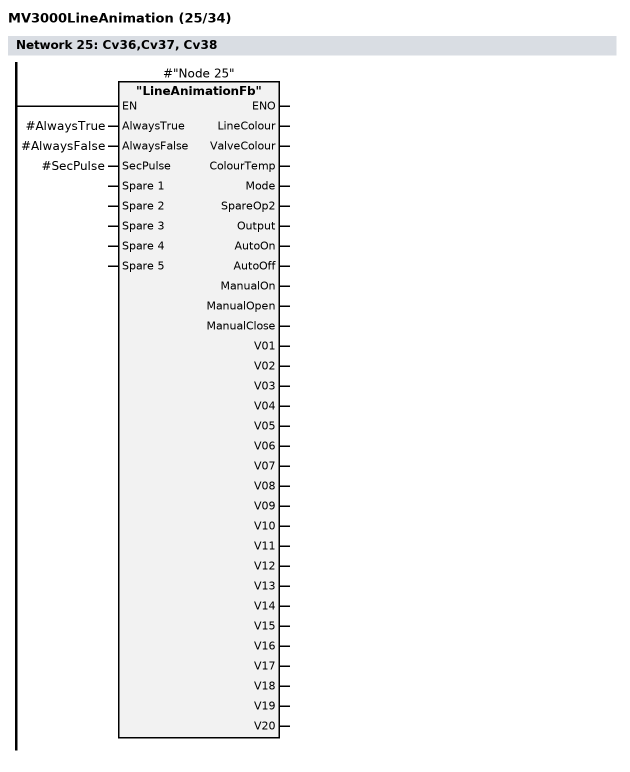
   RUNG wire#powerrail
      #"Node 25"(AlwaysTrue := #AlwaysTrue, AlwaysFalse := #AlwaysFalse, SecPulse := #SecPulse, "Spare 1" :=, "Spare 2" :=, "Spare 3" :=, "Spare 4" :=, "Spare 5" :=, LineColour =>, ValveColour =>, ColourTemp =>, Mode =>, SpareOp2 =>, Output =>, AutoOn =>, AutoOff =>, ManualOn =>, ManualOpen =>, ManualClose =>, V01 =>, V02 =>, V03 =>, V04 =>, V05 =>, V06 =>, V07 =>, V08 =>, V09 =>, V10 =>, V11 =>, V12 =>, V13 =>, V14 =>, V15 =>, V16 =>, V17 =>, V18 =>, V19 =>, V20 =>)
   END_RUNG
   // the same network as SCL:
   #"Node 25"(AlwaysTrue := #AlwaysTrue, AlwaysFalse := #AlwaysFalse, SecPulse := #SecPulse);   // "LineAnimationFb"
END_REGION

REGION Network 26: Cv30,Cv33, Cv34,Cv35
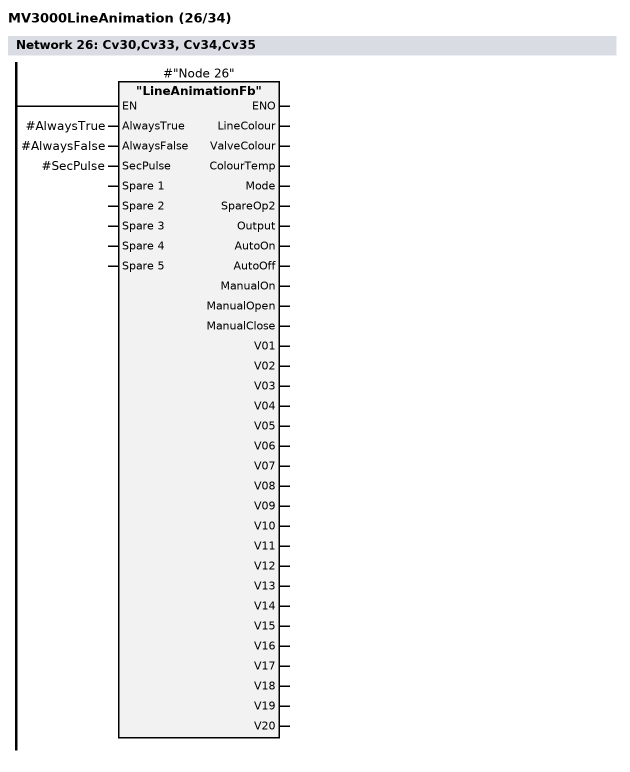
   RUNG wire#powerrail
      #"Node 26"(AlwaysTrue := #AlwaysTrue, AlwaysFalse := #AlwaysFalse, SecPulse := #SecPulse, "Spare 1" :=, "Spare 2" :=, "Spare 3" :=, "Spare 4" :=, "Spare 5" :=, LineColour =>, ValveColour =>, ColourTemp =>, Mode =>, SpareOp2 =>, Output =>, AutoOn =>, AutoOff =>, ManualOn =>, ManualOpen =>, ManualClose =>, V01 =>, V02 =>, V03 =>, V04 =>, V05 =>, V06 =>, V07 =>, V08 =>, V09 =>, V10 =>, V11 =>, V12 =>, V13 =>, V14 =>, V15 =>, V16 =>, V17 =>, V18 =>, V19 =>, V20 =>)
   END_RUNG
   // the same network as SCL:
   #"Node 26"(AlwaysTrue := #AlwaysTrue, AlwaysFalse := #AlwaysFalse, SecPulse := #SecPulse);   // "LineAnimationFb"
END_REGION

REGION Network 27: Cv28, Cv34,Cv37,Cv45,Cv51, Cv57,Cv60
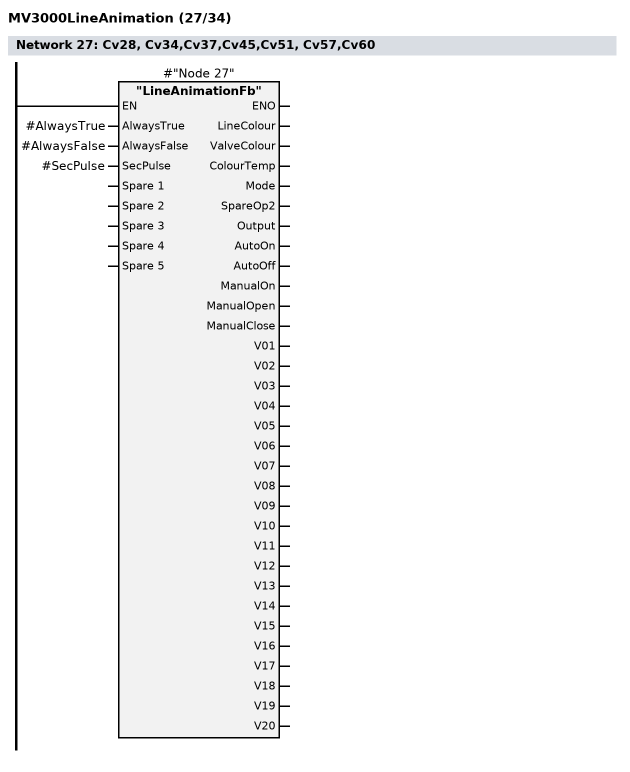
   RUNG wire#powerrail
      #"Node 27"(AlwaysTrue := #AlwaysTrue, AlwaysFalse := #AlwaysFalse, SecPulse := #SecPulse, "Spare 1" :=, "Spare 2" :=, "Spare 3" :=, "Spare 4" :=, "Spare 5" :=, LineColour =>, ValveColour =>, ColourTemp =>, Mode =>, SpareOp2 =>, Output =>, AutoOn =>, AutoOff =>, ManualOn =>, ManualOpen =>, ManualClose =>, V01 =>, V02 =>, V03 =>, V04 =>, V05 =>, V06 =>, V07 =>, V08 =>, V09 =>, V10 =>, V11 =>, V12 =>, V13 =>, V14 =>, V15 =>, V16 =>, V17 =>, V18 =>, V19 =>, V20 =>)
   END_RUNG
   // the same network as SCL:
   #"Node 27"(AlwaysTrue := #AlwaysTrue, AlwaysFalse := #AlwaysFalse, SecPulse := #SecPulse);   // "LineAnimationFb"
END_REGION

REGION Network 28: Cv22, Cv25,Cv19,Cv20,Cv29,Cv35, Cv38,C46 ,Cv52 ,Cv58 ,Cv59
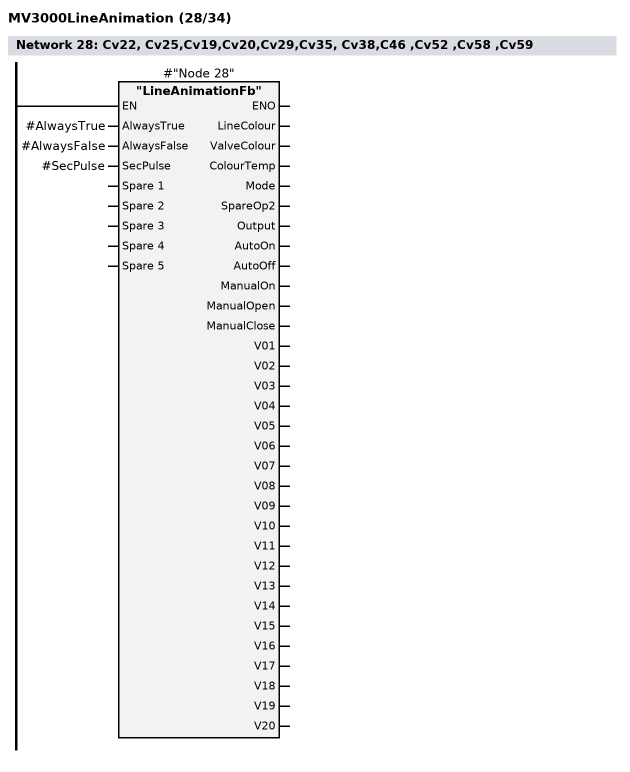
   RUNG wire#powerrail
      #"Node 28"(AlwaysTrue := #AlwaysTrue, AlwaysFalse := #AlwaysFalse, SecPulse := #SecPulse, "Spare 1" :=, "Spare 2" :=, "Spare 3" :=, "Spare 4" :=, "Spare 5" :=, LineColour =>, ValveColour =>, ColourTemp =>, Mode =>, SpareOp2 =>, Output =>, AutoOn =>, AutoOff =>, ManualOn =>, ManualOpen =>, ManualClose =>, V01 =>, V02 =>, V03 =>, V04 =>, V05 =>, V06 =>, V07 =>, V08 =>, V09 =>, V10 =>, V11 =>, V12 =>, V13 =>, V14 =>, V15 =>, V16 =>, V17 =>, V18 =>, V19 =>, V20 =>)
   END_RUNG
   // the same network as SCL:
   #"Node 28"(AlwaysTrue := #AlwaysTrue, AlwaysFalse := #AlwaysFalse, SecPulse := #SecPulse);   // "LineAnimationFb"
END_REGION

REGION Network 29: Cv01,Cv04
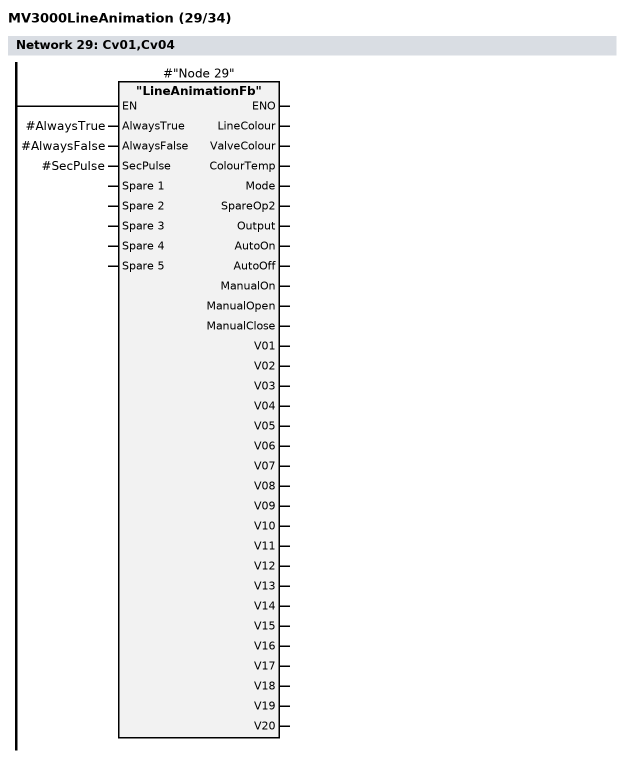
   RUNG wire#powerrail
      #"Node 29"(AlwaysTrue := #AlwaysTrue, AlwaysFalse := #AlwaysFalse, SecPulse := #SecPulse, "Spare 1" :=, "Spare 2" :=, "Spare 3" :=, "Spare 4" :=, "Spare 5" :=, LineColour =>, ValveColour =>, ColourTemp =>, Mode =>, SpareOp2 =>, Output =>, AutoOn =>, AutoOff =>, ManualOn =>, ManualOpen =>, ManualClose =>, V01 =>, V02 =>, V03 =>, V04 =>, V05 =>, V06 =>, V07 =>, V08 =>, V09 =>, V10 =>, V11 =>, V12 =>, V13 =>, V14 =>, V15 =>, V16 =>, V17 =>, V18 =>, V19 =>, V20 =>)
   END_RUNG
   // the same network as SCL:
   #"Node 29"(AlwaysTrue := #AlwaysTrue, AlwaysFalse := #AlwaysFalse, SecPulse := #SecPulse);   // "LineAnimationFb"
END_REGION

REGION Network 30: Cv06,Cv09
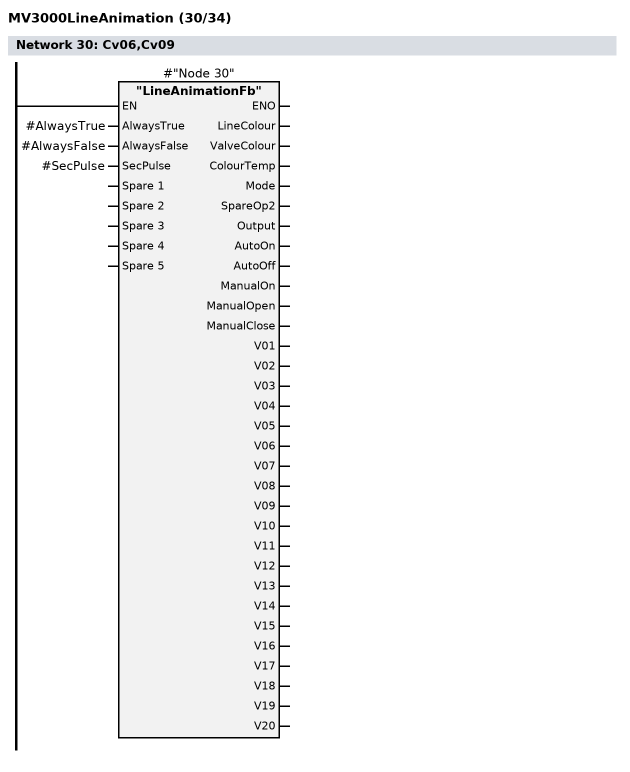
   RUNG wire#powerrail
      #"Node 30"(AlwaysTrue := #AlwaysTrue, AlwaysFalse := #AlwaysFalse, SecPulse := #SecPulse, "Spare 1" :=, "Spare 2" :=, "Spare 3" :=, "Spare 4" :=, "Spare 5" :=, LineColour =>, ValveColour =>, ColourTemp =>, Mode =>, SpareOp2 =>, Output =>, AutoOn =>, AutoOff =>, ManualOn =>, ManualOpen =>, ManualClose =>, V01 =>, V02 =>, V03 =>, V04 =>, V05 =>, V06 =>, V07 =>, V08 =>, V09 =>, V10 =>, V11 =>, V12 =>, V13 =>, V14 =>, V15 =>, V16 =>, V17 =>, V18 =>, V19 =>, V20 =>)
   END_RUNG
   // the same network as SCL:
   #"Node 30"(AlwaysTrue := #AlwaysTrue, AlwaysFalse := #AlwaysFalse, SecPulse := #SecPulse);   // "LineAnimationFb"
END_REGION

REGION Network 31: Cv06,Cv09 ,Cv08
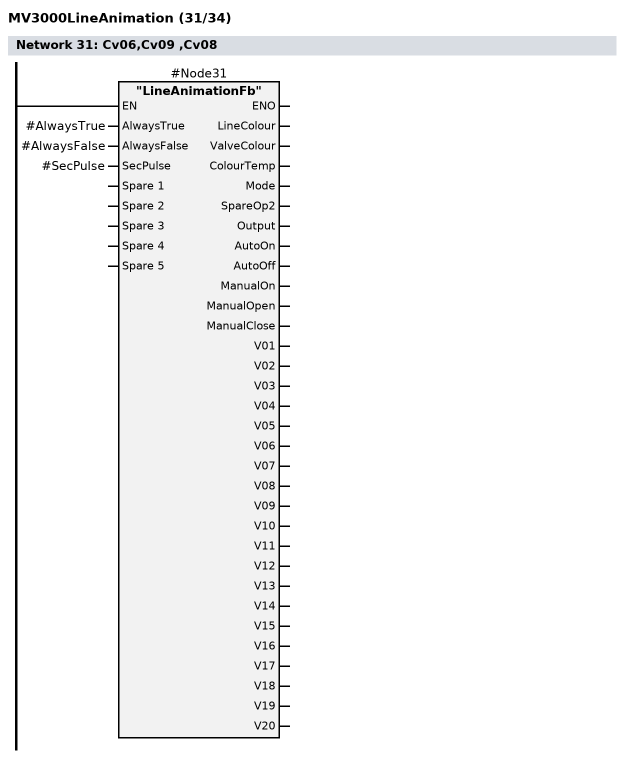
   RUNG wire#powerrail
      #Node31(AlwaysTrue := #AlwaysTrue, AlwaysFalse := #AlwaysFalse, SecPulse := #SecPulse, "Spare 1" :=, "Spare 2" :=, "Spare 3" :=, "Spare 4" :=, "Spare 5" :=, LineColour =>, ValveColour =>, ColourTemp =>, Mode =>, SpareOp2 =>, Output =>, AutoOn =>, AutoOff =>, ManualOn =>, ManualOpen =>, ManualClose =>, V01 =>, V02 =>, V03 =>, V04 =>, V05 =>, V06 =>, V07 =>, V08 =>, V09 =>, V10 =>, V11 =>, V12 =>, V13 =>, V14 =>, V15 =>, V16 =>, V17 =>, V18 =>, V19 =>, V20 =>)
   END_RUNG
   // the same network as SCL:
   #Node31(AlwaysTrue := #AlwaysTrue, AlwaysFalse := #AlwaysFalse, SecPulse := #SecPulse);   // "LineAnimationFb"
END_REGION

REGION Network 32: Cv05,Cv24
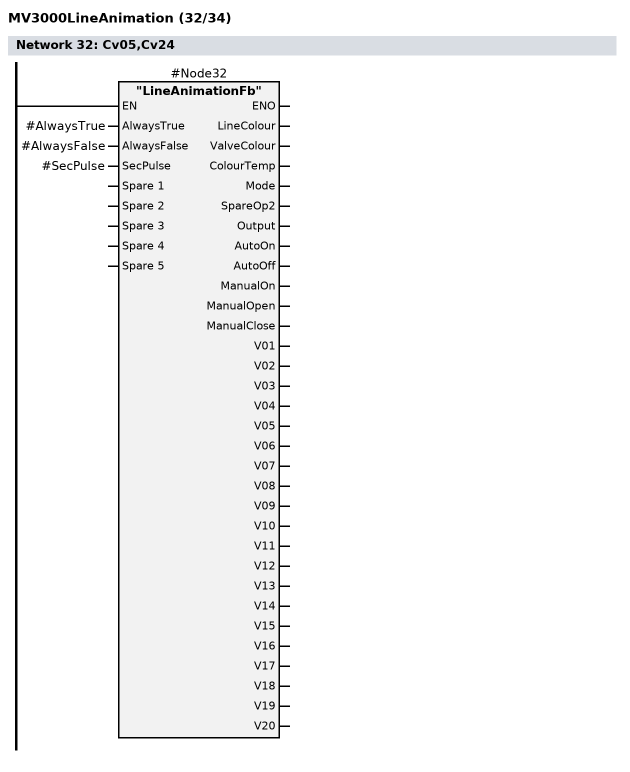
   RUNG wire#powerrail
      #Node32(AlwaysTrue := #AlwaysTrue, AlwaysFalse := #AlwaysFalse, SecPulse := #SecPulse, "Spare 1" :=, "Spare 2" :=, "Spare 3" :=, "Spare 4" :=, "Spare 5" :=, LineColour =>, ValveColour =>, ColourTemp =>, Mode =>, SpareOp2 =>, Output =>, AutoOn =>, AutoOff =>, ManualOn =>, ManualOpen =>, ManualClose =>, V01 =>, V02 =>, V03 =>, V04 =>, V05 =>, V06 =>, V07 =>, V08 =>, V09 =>, V10 =>, V11 =>, V12 =>, V13 =>, V14 =>, V15 =>, V16 =>, V17 =>, V18 =>, V19 =>, V20 =>)
   END_RUNG
   // the same network as SCL:
   #Node32(AlwaysTrue := #AlwaysTrue, AlwaysFalse := #AlwaysFalse, SecPulse := #SecPulse);   // "LineAnimationFb"
END_REGION

REGION Network 33: CvFbv01,Cv26
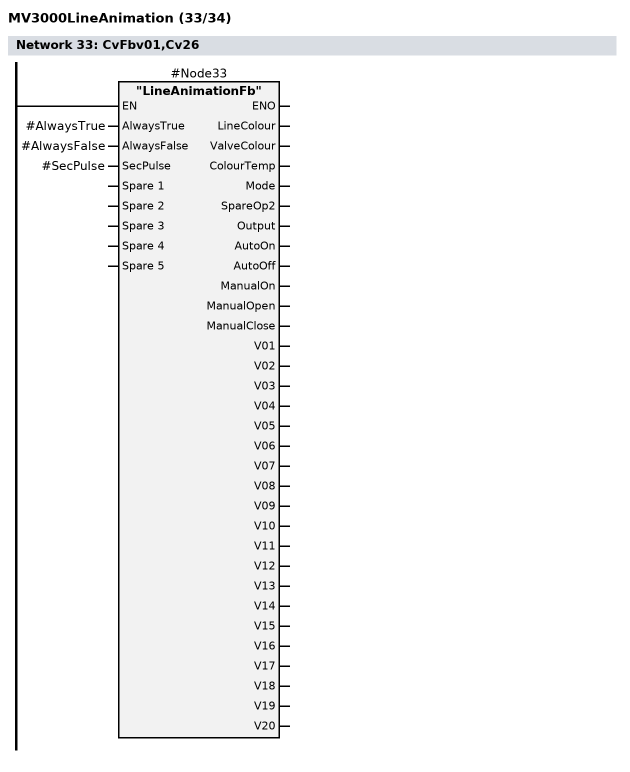
   RUNG wire#powerrail
      #Node33(AlwaysTrue := #AlwaysTrue, AlwaysFalse := #AlwaysFalse, SecPulse := #SecPulse, "Spare 1" :=, "Spare 2" :=, "Spare 3" :=, "Spare 4" :=, "Spare 5" :=, LineColour =>, ValveColour =>, ColourTemp =>, Mode =>, SpareOp2 =>, Output =>, AutoOn =>, AutoOff =>, ManualOn =>, ManualOpen =>, ManualClose =>, V01 =>, V02 =>, V03 =>, V04 =>, V05 =>, V06 =>, V07 =>, V08 =>, V09 =>, V10 =>, V11 =>, V12 =>, V13 =>, V14 =>, V15 =>, V16 =>, V17 =>, V18 =>, V19 =>, V20 =>)
   END_RUNG
   // the same network as SCL:
   #Node33(AlwaysTrue := #AlwaysTrue, AlwaysFalse := #AlwaysFalse, SecPulse := #SecPulse);   // "LineAnimationFb"
END_REGION

REGION Network 34: Cv42,Cv54,Cv48
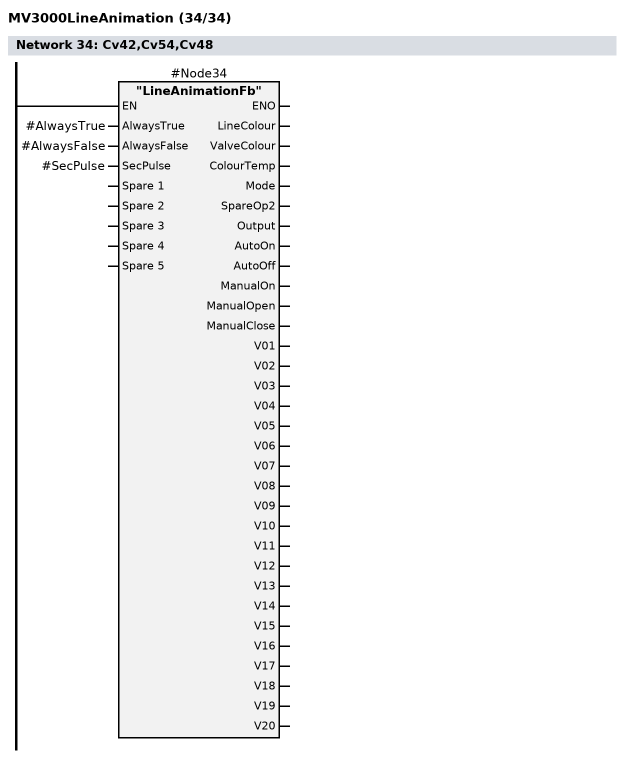
   RUNG wire#powerrail
      #Node34(AlwaysTrue := #AlwaysTrue, AlwaysFalse := #AlwaysFalse, SecPulse := #SecPulse, "Spare 1" :=, "Spare 2" :=, "Spare 3" :=, "Spare 4" :=, "Spare 5" :=, LineColour =>, ValveColour =>, ColourTemp =>, Mode =>, SpareOp2 =>, Output =>, AutoOn =>, AutoOff =>, ManualOn =>, ManualOpen =>, ManualClose =>, V01 =>, V02 =>, V03 =>, V04 =>, V05 =>, V06 =>, V07 =>, V08 =>, V09 =>, V10 =>, V11 =>, V12 =>, V13 =>, V14 =>, V15 =>, V16 =>, V17 =>, V18 =>, V19 =>, V20 =>)
   END_RUNG
   // the same network as SCL:
   #Node34(AlwaysTrue := #AlwaysTrue, AlwaysFalse := #AlwaysFalse, SecPulse := #SecPulse);   // "LineAnimationFb"
END_REGION
END_FUNCTION_BLOCK
